FUNCTION_BLOCK StandardRoom IMPLEMENTS I_Execute, I_Init
VAR_INPUT
	rTemperature	: LREAL := 20.0 + Random();
	
	bInletValveIsClosed	: BOOL;
	bInletValveIsOpen	: BOOL;
	
	bOutletValveIsClosed: BOOL;
	bOutletValveIsOpen	: BOOL;
END_VAR
VAR_OUTPUT
	bInletValve		: BOOL;
	bOutletValve	: BOOL;
END_VAR
VAR	
	
	// Entity declaration, context and execute
	_this			: Entity;
	_ctx			: Room_Ctx;
	_tag			: Tag(CONCAT('Room_', UDINT_TO_STRING(_ctx.Id)));
	_compTag		: Comp(_tag, _this);
	_exe			: Execute(THIS^);
	_init			: Init(THIS^);
	
	// UI Logic
	_uiLogic		: Room_UiLogic(_ctx);
	
	// Receiver
	_onSystemEvent	: Room_OnSystemEvent(_ctx);
	
	// Signal
	_requestEvent		: Signal;
	_compRequestEvent	: Comp(_requestEvent, _this);
	_proxRequestEvent	: SignalProxy(_requestEvent, _ctx.priv.iRequestEvent);
	
	
	// State Manager
	_smgr			: StateManager(_this);
	_proxSmgr		: StateManagerProxy(_smgr, _ctx.state.iMgr);
	
	// States
	_disable		: Room_State_Disabled(_this, _ctx);
	_proxDisable	: StateProxy(_disable, _ctx.state.iDisable);
	
	_fault			: Room_State_Fault(_this,_ctx);
	_proxFault		: StateProxy(_fault, _ctx.state.iFault);	
	
	_idle			: Room_State_Idle(_this,_ctx);
	_proxIdle		: StateProxy(_idle, _ctx.state.iIdle);
	
	_lowTemperature	: Room_State_LowTemperature(_this, _ctx, rTemperature);
	
	_demand			: Room_State_DemandHeating(_this, _ctx);
	
	
	// Simulation
	_inletSim		: ValveSim(bInletValve, bInletValveIsOpen, bInletValveIsClosed);
	_outletSim		: ValveSim(bOutletValve, bOutletValveIsOpen, bOutletValveIsClosed);
		
END_VAR

METHOD Execute
// HMI

_ctx.hmi.sData := '';

// Inputs
_ctx.io.bValvesOpen := bInletValveIsOpen AND bOutletValveIsOpen;
_ctx.io.bValvesClosed := bInletValveIsClosed AND bOutletValveIsClosed;

// Outputs
bInletValve := _ctx.io.bOpenValves;
bOutletValve := _ctx.io.bOpenValves;

// Simulation
IF NOT sim.bTick THEN
	RETURN;
END_IF

IF bInletValve AND bOutletValve THEN
	sim.rSystemTemperature := sim.rSystemTemperature + sim.param.rSystemTemperatureDropPerHeater * Random();
	rTemperature := rTemperature + sim.param.rRoomTemperatureRisePerHeater * Random();
END_IF

rTemperature := rTemperature + sim.param.rRoomTemperaturePassiveDrop * Random();

IF rTemperature < 0 THEN
	rTemperature := 0;
ELSIF rTemperature > 100 THEN
	rTemperature := 100;
END_IF
END_METHOD

METHOD Init
_smgr.Request(_idle);
END_METHOD

END_FUNCTION_BLOCK

(* stored: Version 1.1.0.1
   POU StandardRoom: Id {2e0e75c6-de15-4761-ae40-14041f36bdf4}, SpecialFunc None
   Method Execute: Id {51b956d4-c76f-41de-a458-174fed593c72}
   Method Init: Id {3ff82767-55bc-4f86-a241-d582f5293491} *)
